FUNCTION_BLOCK fb_gm_operationSV
VAR_INPUT
END_VAR
VAR_OUTPUT
END_VAR
VAR
	trn_gm_chuckOpenDone: BOOL;
	trn_gm_chuckCloseDone: BOOL;
	trn_gm_pushCloseDone: BOOL;
	trn_gm_pushOpenDone: BOOL;
	trn_gm_rotaryOriginDone: BOOL;
	trn_gm_rotaryMovingDone: BOOL;
	trn_gm_pickUpOriginDone: BOOL;
	trn_gm_pickUpMovingDone: BOOL;
	trn_gm_stampOriginDone: BOOL;
	trn_gm_stampMovingDone: BOOL;
	trn_flgInitDone: BOOL;
	flg_test: BOOL;
	flg_test2: BOOL;
END_VAR

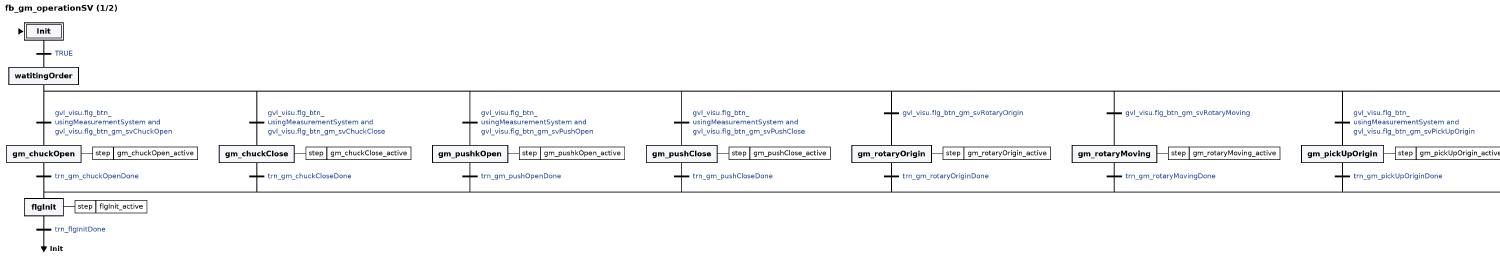
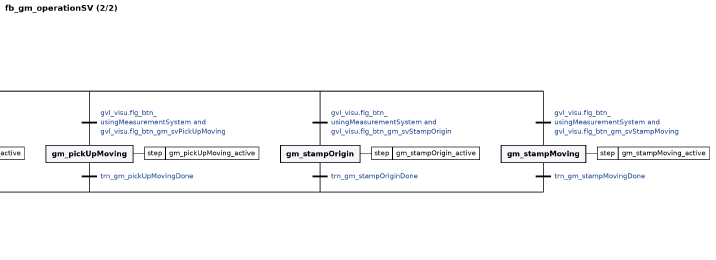
INITIAL_STEP Init:
END_STEP
TRANSITION FROM Init TO watitingOrder
    := TRUE;
END_TRANSITION
STEP watitingOrder:
END_STEP
TRANSITION FROM watitingOrder TO gm_chuckOpen
    := gvl_visu.flg_btn_usingMeasurementSystem and gvl_visu.flg_btn_gm_svChuckOpen;
END_TRANSITION
STEP gm_chuckOpen:
    gm_chuckOpen_active(N);  // step action
END_STEP
TRANSITION FROM gm_chuckOpen TO flgInit
    := trn_gm_chuckOpenDone;
END_TRANSITION
TRANSITION FROM watitingOrder TO gm_chuckClose
    := gvl_visu.flg_btn_usingMeasurementSystem and gvl_visu.flg_btn_gm_svChuckClose;
END_TRANSITION
STEP gm_chuckClose:
    gm_chuckClose_active(N);  // step action
END_STEP
TRANSITION FROM gm_chuckClose TO flgInit
    := trn_gm_chuckCloseDone;
END_TRANSITION
TRANSITION FROM watitingOrder TO gm_pushkOpen
    := gvl_visu.flg_btn_usingMeasurementSystem and gvl_visu.flg_btn_gm_svPushOpen;
END_TRANSITION
STEP gm_pushkOpen:
    gm_pushkOpen_active(N);  // step action
END_STEP
TRANSITION FROM gm_pushkOpen TO flgInit
    := trn_gm_pushOpenDone;
END_TRANSITION
TRANSITION FROM watitingOrder TO gm_pushClose
    := gvl_visu.flg_btn_usingMeasurementSystem and gvl_visu.flg_btn_gm_svPushClose;
END_TRANSITION
STEP gm_pushClose:
    gm_pushClose_active(N);  // step action
END_STEP
TRANSITION FROM gm_pushClose TO flgInit
    := trn_gm_pushCloseDone;
END_TRANSITION
TRANSITION FROM watitingOrder TO gm_rotaryOrigin
    := gvl_visu.flg_btn_gm_svRotaryOrigin;
END_TRANSITION
STEP gm_rotaryOrigin:
    gm_rotaryOrigin_active(N);  // step action
END_STEP
TRANSITION FROM gm_rotaryOrigin TO flgInit
    := trn_gm_rotaryOriginDone;
END_TRANSITION
TRANSITION FROM watitingOrder TO gm_rotaryMoving
    := gvl_visu.flg_btn_gm_svRotaryMoving;
END_TRANSITION
STEP gm_rotaryMoving:
    gm_rotaryMoving_active(N);  // step action
END_STEP
TRANSITION FROM gm_rotaryMoving TO flgInit
    := trn_gm_rotaryMovingDone;
END_TRANSITION
TRANSITION FROM watitingOrder TO gm_pickUpOrigin
    := gvl_visu.flg_btn_usingMeasurementSystem and gvl_visu.flg_btn_gm_svPickUpOrigin;
END_TRANSITION
STEP gm_pickUpOrigin:
    gm_pickUpOrigin_active(N);  // step action
END_STEP
TRANSITION FROM gm_pickUpOrigin TO flgInit
    := trn_gm_pickUpOriginDone;
END_TRANSITION
TRANSITION FROM watitingOrder TO gm_pickUpMoving
    := gvl_visu.flg_btn_usingMeasurementSystem and gvl_visu.flg_btn_gm_svPickUpMoving;
END_TRANSITION
STEP gm_pickUpMoving:
    gm_pickUpMoving_active(N);  // step action
END_STEP
TRANSITION FROM gm_pickUpMoving TO flgInit
    := trn_gm_pickUpMovingDone;
END_TRANSITION
TRANSITION FROM watitingOrder TO gm_stampOrigin
    := gvl_visu.flg_btn_usingMeasurementSystem and gvl_visu.flg_btn_gm_svStampOrigin;
END_TRANSITION
STEP gm_stampOrigin:
    gm_stampOrigin_active(N);  // step action
END_STEP
TRANSITION FROM gm_stampOrigin TO flgInit
    := trn_gm_stampOriginDone;
END_TRANSITION
TRANSITION FROM watitingOrder TO gm_stampMoving
    := gvl_visu.flg_btn_usingMeasurementSystem and gvl_visu.flg_btn_gm_svStampMoving;
END_TRANSITION
STEP gm_stampMoving:
    gm_stampMoving_active(N);  // step action
END_STEP
TRANSITION FROM gm_stampMoving TO flgInit
    := trn_gm_stampMovingDone;
END_TRANSITION
STEP flgInit:
    flgInit_active(N);  // step action
END_STEP
TRANSITION FROM flgInit TO Init
    := trn_flgInitDone;
END_TRANSITION

ACTION flgInit_active:
IF flgInit._x AND flgInit.x = FALSE THEN
	trn_flgInitDone := FALSE;
	gvl_visu.flg_btn_gm_svChuckOpen := FALSE;
	gvl_visu.flg_btn_gm_svChuckClose := FALSE;
	gvl_visu.flg_btn_gm_svPushOpen := FALSE;
	gvl_visu.flg_btn_gm_svPushClose := FALSE;
	gvl_visu.flg_btn_gm_svRotaryOrigin := FALSE;
	gvl_visu.flg_btn_gm_svRotaryMoving := FALSE;
	gvl_visu.flg_btn_gm_svPickUpOrigin := FALSE;
	gvl_visu.flg_btn_gm_svPickUpMoving := FALSE;
	gvl_visu.flg_btn_gm_svStampOrigin := FALSE;
	gvl_visu.flg_btn_gm_svStampMoving := FALSE;
ELSIF flgInit._x AND flgInit.x THEN
	trn_flgInitDone := TRUE;
END_IF
END_ACTION

ACTION gm_chuckClose_active:
IF gm_chuckClose._x AND gm_chuckClose.x = FALSE THEN
	trn_gm_chuckCloseDone := FALSE;
	gvl_solv.fbi_gm_chuck.in_flg_run := FALSE;
	gvl_solv.fbi_gm_chuck.in_var_moveMode := eP_svMoveMode.svB;
ELSIF gm_chuckClose._x AND gm_chuckClose.x THEN
	gvl_solv.fbi_gm_chuck.in_flg_run := TRUE;
	IF gvl_solv.fbi_gm_chuck.out_flg_Done THEN
		gvl_solv.fbi_gm_chuck.in_flg_run := FALSE;
		trn_gm_chuckCloseDone := TRUE;
	END_IF
END_IF
END_ACTION

ACTION gm_chuckOpen_active:
IF gm_chuckOpen._x AND gm_chuckOpen.x = FALSE THEN
	trn_gm_chuckOpenDone := FALSE;
	gvl_solv.fbi_gm_chuck.in_flg_run := FALSE;
	gvl_solv.fbi_gm_chuck.in_var_moveMode := eP_svMoveMode.svA;
ELSIF gm_chuckOpen._x AND gm_chuckOpen.x THEN
	gvl_solv.fbi_gm_chuck.in_flg_run := TRUE;
	IF gvl_solv.fbi_gm_chuck.out_flg_Done THEN
		gvl_solv.fbi_gm_chuck.in_flg_run := FALSE;
		trn_gm_chuckOpenDone := TRUE;
	END_IF
END_IF
END_ACTION

ACTION gm_pickUpMoving_active:
IF gm_pickUpMoving._x AND gm_pickUpMoving.x = FALSE THEN
	trn_gm_pickUpMovingDone := FALSE;
	gvl_solv.fbi_gm_pickup.in_flg_run := FALSE;
	gvl_solv.fbi_gm_pickup.in_var_moveMode := eP_svMoveMode.svB;
ELSIF gm_pickUpMoving._x AND gm_pickUpMoving.x THEN
		gvl_solv.fbi_gm_pickup.in_flg_run := TRUE;
	IF gvl_solv.fbi_gm_pickup.out_flg_Done THEN
		gvl_solv.fbi_gm_pickup.in_flg_run := FALSE;
		trn_gm_pickUpMovingDone := TRUE;
	END_IF
END_IF
END_ACTION

ACTION gm_pickUpOrigin_active:
IF gm_pickUpOrigin._x AND gm_pickUpOrigin.x = FALSE THEN
	trn_gm_pickUpOriginDone := FALSE;
	gvl_solv.fbi_gm_pickup.in_flg_run := FALSE;
	gvl_solv.fbi_gm_pickup.in_var_moveMode := eP_svMoveMode.svA;
ELSIF gm_pickUpOrigin._x AND gm_pickUpOrigin.x THEN
		gvl_solv.fbi_gm_pickup.in_flg_run := TRUE;
	IF gvl_solv.fbi_gm_pickup.out_flg_Done THEN
		gvl_solv.fbi_gm_pickup.in_flg_run := FALSE;
		trn_gm_pickUpOriginDone := TRUE;
	END_IF
END_IF
END_ACTION

ACTION gm_pushClose_active:
IF gm_pushClose._x AND gm_pushClose.x = FALSE THEN
	trn_gm_pushCloseDone := FALSE;
	gvl_solv.fbi_gm_push.in_flg_run := FALSE;
	gvl_solv.fbi_gm_push.in_var_moveMode := eP_svMoveMode.svB;
ELSIF gm_pushClose._x AND gm_pushClose.x THEN
	gvl_solv.fbi_gm_push.in_flg_run := TRUE;
	IF gvl_solv.fbi_gm_push.out_flg_Done THEN
		gvl_solv.fbi_gm_push.in_flg_run := FALSE;
		trn_gm_pushCloseDone := TRUE;
	END_IF
END_IF
END_ACTION

ACTION gm_pushkOpen_active:
IF gm_pushkOpen._x AND gm_pushkOpen.x = FALSE THEN
	trn_gm_pushOpenDone := FALSE;
	gvl_solv.fbi_gm_push.in_flg_run := FALSE;
	gvl_solv.fbi_gm_push.in_var_moveMode := eP_svMoveMode.svA;
ELSIF gm_pushkOpen._x AND gm_pushkOpen.x THEN
	gvl_solv.fbi_gm_push.in_flg_run := TRUE;
	IF gvl_solv.fbi_gm_push.out_flg_Done THEN
 		gvl_solv.fbi_gm_push.in_flg_run := FALSE;
		trn_gm_pushOpenDone := TRUE;
	END_IF
END_IF
END_ACTION

ACTION gm_rotaryMoving_active:
IF gm_rotaryMoving._x AND gm_rotaryMoving.x = FALSE THEN
	trn_gm_rotaryMovingDone := FALSE;
	gvl_solv.fbi_gm_rotary.in_flg_run := FALSE;
	gvl_solv.fbi_gm_rotary.in_var_moveMode := eP_svMoveMode.svB;
ELSIF gm_rotaryMoving._x AND gm_rotaryMoving.x THEN
		gvl_solv.fbi_gm_rotary.in_flg_run := TRUE;
	IF gvl_solv.fbi_gm_rotary.out_flg_Done THEN
		gvl_solv.fbi_gm_rotary.in_flg_run := FALSE;
		trn_gm_rotaryMovingDone := TRUE;
	END_IF
END_IF
END_ACTION

ACTION gm_rotaryOrigin_active:
IF gm_rotaryOrigin._x AND gm_rotaryOrigin.x = FALSE THEN
	trn_gm_rotaryOriginDone := FALSE;
	gvl_solv.fbi_gm_rotary.in_flg_run := FALSE;
	gvl_solv.fbi_gm_rotary.in_var_moveMode := eP_svMoveMode.svA;
ELSIF gm_rotaryOrigin._x AND gm_rotaryOrigin.x THEN
	gvl_solv.fbi_gm_rotary.in_flg_run := TRUE;
	IF gvl_solv.fbi_gm_rotary.out_flg_Done THEN
		gvl_solv.fbi_gm_rotary.in_flg_run := FALSE;
		trn_gm_rotaryOriginDone := TRUE;
	END_IF
END_IF
END_ACTION

ACTION gm_stampMoving_active:
IF gm_stampMoving._x AND gm_stampMoving.x = FALSE THEN
	trn_gm_stampMovingDone := FALSE;
	gvl_solv.fbi_gm_stamp.in_flg_run := FALSE;
	gvl_solv.fbi_gm_stamp.in_var_moveMode := eP_svMoveMode.svB;
ELSIF gm_stampMoving._x AND gm_stampMoving.x THEN
		gvl_solv.fbi_gm_stamp.in_flg_run := TRUE;
	IF gvl_solv.fbi_gm_stamp.out_flg_Done THEN
		gvl_solv.fbi_gm_stamp.in_flg_run := FALSE;
		trn_gm_stampMovingDone := TRUE;
	END_IF
END_IF
END_ACTION

ACTION gm_stampOrigin_active:
IF gm_stampOrigin._x AND gm_stampOrigin.x = FALSE THEN
	trn_gm_stampOriginDone := FALSE;
	gvl_solv.fbi_gm_stamp.in_flg_run := FALSE;
	gvl_solv.fbi_gm_stamp.in_var_moveMode := eP_svMoveMode.svA;
ELSIF gm_stampOrigin._x AND gm_stampOrigin.x THEN
		gvl_solv.fbi_gm_stamp.in_flg_run := TRUE;
	IF gvl_solv.fbi_gm_stamp.out_flg_Done THEN
		gvl_solv.fbi_gm_stamp.in_flg_run := FALSE;
		trn_gm_stampOriginDone := TRUE;
	END_IF
END_IF
END_ACTION

PROPERTY p_Init : bool
GET
p_init := THIS^.SFCInit;
END_GET
SET
THIS^.SFCInit := p_init;
END_SET
END_PROPERTY

END_FUNCTION_BLOCK

(* stored: Version 1.1.0.1, ProductVersion 3.1.4024.11
   POU fb_gm_operationSV: Id {70ad780b-e8ad-4dde-8431-67951edc7fb4}, SpecialFunc None
   Action flgInit_active: Id {131f28c1-ec80-48d9-bb2d-0a2b4bd1e3fc}
   Action gm_chuckClose_active: Id {6900e230-c4a6-48c6-8361-a11f83b24c15}
   Action gm_chuckOpen_active: Id {df11605c-ccb1-4101-beb7-408601c1c460}
   Action gm_pickUpMoving_active: Id {daf8d92f-4863-485a-a227-56fe21fa8241}
   Action gm_pickUpOrigin_active: Id {4d0bc22e-e0b1-4bd2-89b7-303c3553b836}
   Action gm_pushClose_active: Id {f2fbf4e5-53cd-4a63-91b7-7b1a1e69a715}
   Action gm_pushkOpen_active: Id {6691f2c0-0ad6-430f-a0ed-d166f5342f12}
   Action gm_rotaryMoving_active: Id {a48a0252-7526-49e5-9dad-4974ea471027}
   Action gm_rotaryOrigin_active: Id {5ddc0da1-34a8-46da-9286-4e4213106cbf}
   Action gm_stampMoving_active: Id {f53c77a1-60d3-4187-87b8-a6d56e5030c6}
   Action gm_stampOrigin_active: Id {7a563519-5412-428b-ad37-8a85408e1976}
   Property p_Init: Id {4e47238c-5790-42d8-bb0f-1db4874c3134}
   Get Get: Id {418d3a4e-2f51-4fbf-bedf-113f8f528b65}
   Set Set: Id {bc6cd654-57c7-4cab-8421-b7a91cf72898} *)
